# EPICS substitutions: GSpiApp/Db/asynRecord.substitutions
file asynRecord.template
{
	pattern { P	     , R		, PORT	, ADDR , OMAX , IMAX }
		{ XF:11ID-M3 , "{Hyrel:1}Asyn"	, HYREL	, 0    , 0    , 0    }
}
